// TwinCAT 3 PLC project Main
// ProgramVersion: 3.1.4023.0
// libraries:
//   Tc2_MC2, * (Beckhoff Automation GmbH)
//   Tc2_Standard, * (Beckhoff Automation GmbH)
//   Tc2_System, * (Beckhoff Automation GmbH)
//   Tc3_Module, * (Beckhoff Automation GmbH)
// project tree:
//   DUTs/Control/ ForceControlParam.TcDUT (not stored), JogParam.TcDUT (not stored)
//   DUTs/ MotorParam.TcDUT, MotorState.TcDUT (not stored), SystemControlMode.TcDUT (not stored), SystemControlParam.TcDUT
//   GVLs/ GVL.TcGVL (not stored)
//   / PlcTask.TcTTO
//   POUs/ MAIN.TcPOU, SystemControl.TcPOU
//   POUs/Safety/ VelocitySaturation.TcPOU
//   POUs/Converter/ CableVelocityToMotorAngularVelocity.TcPOU, MotorAngularVelocityToCableVelocity.TcPOU, MotorDegreeToCablePosition.TcPOU (not stored)
// real-time tasks:
//   TASK PlcTask: cycle T#10ms, priority 20, ADS port 350
// motion (NC):
//   TASK NC-Task 1 SAF: cycle T#2ms, priority 4, ADS port 501
//   TASK NC-Task 1 SVB: cycle T#10ms, priority 8, ADS port 511
//   AXIS Axis 1 (id 1)
//     General: UnitName=Degree
//     Dynamic: Acceleration=1080, Deceleration=1080, Jerk=3240
//     Velo: RefSearch=180, RefSync=180, SlowManual=180, FastManual=360, Fast=18075.9448242188, Maximum=720
//     PositionAreaControl: Enable=false
//     TargetPosControl: Enable=false
//     OtherSettings: AllowMotionCmdToSlave=true
//     encoder EncType=8
//       EncPara: ScaleFactorNumerator=360, ScaleFactorDenominator=1048576, MaxCount=#xffffffff
//     drive DrvType=9
//       DrvPara: MaxCount=#xffffffff, DriveControlDWord=#x00000100
//         Analog: VeloReferenz=360, VeloScale=1.02400649589962, TorqueSetpointScale=10, ScaleFactorActTorque=0.1
//         TimeComp: TaskDelayCycles=1
//     controller CtrType=1
//       CtrPara: PriorControlFactor=1
//         PosDiffControl: Enable=false
//         Observer: BandWidth=20
// I/O:
//   DEVICE Device 3 (EtherCAT), AmsNetId 192.168.137.1.4.1
//     Term 1 (EK1100) [EK1100 EtherCAT Coupler (2A E-Bus)]
//       Term 2 (EL9505) [EL9505 Power supply terminal 5V]
//       Term 3 (EL3356) [EL3356 1Ch. Ana. Input Resistor Bridge Terminal, 16bit, High Precision]
//       Term 5 (EL9011) [EL9011 End Terminal]
//     Drive 4 (AX5106-0000-0203) [AX5106-0000-0203 EtherCAT Drive (SoE, 1 Ch.)]
// variable links:
//   NC-Task 1 SAF/Axes/Axis 1 <-> Device 3 (EtherCAT)/Drive 4 (AX5106-0000-0203)
//     Drive/Inputs/In/nDcOutputTime <-> InfoData/DcOutputShift
//     Drive/Inputs/In/nState1 <-> AT/Drive status word @bit 8
//     Drive/Inputs/In/nState2 <-> AT/Drive status word
//     Drive/Inputs/In/nState4 @bit 1 <-> WcState/InputToggle
//     Drive/Inputs/In/nState4 <-> WcState/WcState
//     Drive/Outputs/Out/nCtrl1 <-> MDT/Master control word @bit 8
//     Enc/Inputs/In/nDcInputTime <-> InfoData/DcInputShift
//     Enc/Inputs/In/nState4 @bit 1 <-> WcState/InputToggle
//     Enc/Inputs/In/nState4 <-> WcState/WcState

CONFIGURATION Main
    RESOURCE PLC ON TwinCAT3
        TASK PlcTask(INTERVAL := T#10ms, PRIORITY := 20);
        PROGRAM MAIN WITH PlcTask : MAIN;
    END_RESOURCE
END_CONFIGURATION

// ---- DUTs/MotorParam.TcDUT
TYPE MotorParam :
STRUCT
	// 发送给电机的速度
	target_axis_velocity_raw : LREAL;
	
	// 期望的放绳速度
	target_cable_velocity : LREAL;
	
	// 最大最小速度(mm/s)
	max_cable_velocity : LREAL := 1000;
	min_cable_velocity : LREAL := -1000;
END_STRUCT
END_TYPE

// ---- DUTs/SystemControlParam.TcDUT
TYPE SystemControlParam :
STRUCT
	is_motor_poweron : BOOL;
	is_system_exit : BOOL;
	is_system_control : BOOL;
	system_control_mode : SystemControlMode;
	
	// Debug
	is_motor_jog : BOOL;
	jog_param : JogParam;
	// ConstForce
	is_force_control : BOOL;
	force_control_param : ForceControlParam;
END_STRUCT
END_TYPE

// ---- POUs/MAIN.TcPOU
PROGRAM MAIN
VAR
	SystemControl : SystemControl;
	
	system_control_param : SystemControlParam;
	motor_state : MotorState;
	motor_param : MotorParam;
END_VAR

// 系统状态读取
GVL.axis1.ReadStatus();
motor_state.is_motor_closedloop := GVL.axis1.Status.ControlLoopClosed;
motor_state.axis_position_raw := GVL.axis1.NcToPlc.ActPos;
motor_state.axis_velocity_raw := GVL.axis1.NcToPlc.ActVelo;

// 电机参数转换
MotorDegreeToCablePosition(motor_position:= motor_state.axis_position_raw, cable_position=> motor_state.cable_position);
MotorAngularVelocityToCableVelocity(motor_velocity:= motor_state.axis_velocity_raw, cable_velocity=> motor_state.cable_velocity);

// 控制状态机
SystemControl(
	motor_axis:= GVL.axis1, 
	system_control_param:= system_control_param, 
	motor_state:= motor_state, 
	target_velocity=> motor_param.target_cable_velocity);

// 安全限制 
VelocitySaturation(
	velocity:= motor_param.target_cable_velocity, 
	max_velocity:= motor_param.max_cable_velocity, 
	min_velocity:= motor_param.min_cable_velocity);

// 电机参数转换
CableVelocityToMotorAngularVelocity(cable_velocity:= motor_param.target_cable_velocity, motor_velocity=> motor_param.target_axis_velocity_raw);

END_PROGRAM

// ---- POUs/SystemControl.TcPOU
FUNCTION_BLOCK SystemControl
VAR_IN_OUT
	motor_axis : Tc2_MC2.AXIS_REF;
	system_control_param : SystemControlParam;
	motor_state : MotorState;
END_VAR
VAR_OUTPUT
	target_velocity : LREAL;
END_VAR
VAR
	motorPower : Tc2_MC2.MC_Power;
END_VAR

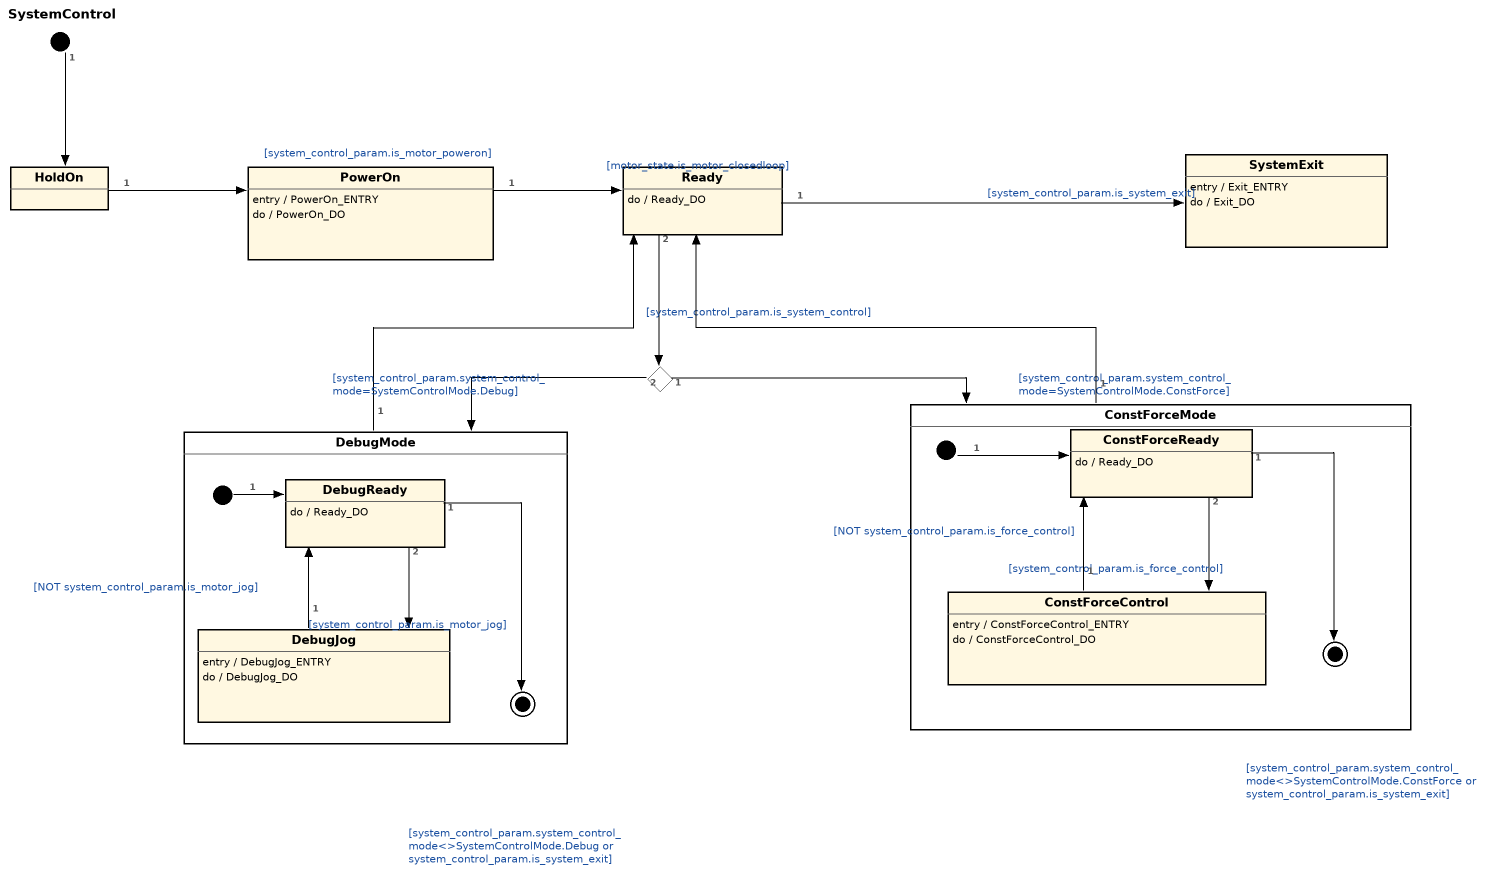
STATECHART SystemControl  // abortable
    START StartState1
    STATE HoldOn
    STATE PowerOn
        entry / PowerOn_ENTRY
        do / PowerOn_DO
    STATE Ready
        do / Ready_DO
    STATE SystemExit
        entry / Exit_ENTRY
        do / Exit_DO
    CHOICE ChoiceElement1
    COMPOSITE STATE ConstForceMode
        START StartState3
        STATE ConstForceReady
            do / Ready_DO
        STATE ConstForceControl
            entry / ConstForceControl_ENTRY
            do / ConstForceControl_DO
        END EndState2
        StartState3 -> ConstForceReady  // priority 1, on completion
        ConstForceReady -> EndState2 [system_control_param.system_control_mode<>SystemControlMode.ConstForce or system_control_param.is_system_exit] // priority 1
        ConstForceReady -> ConstForceControl [system_control_param.is_force_control] // priority 2
        ConstForceControl -> ConstForceReady [NOT system_control_param.is_force_control] // priority 1
    END_STATE
    COMPOSITE STATE DebugMode
        START StartState2
        STATE DebugReady
            do / Ready_DO
        STATE DebugJog
            entry / DebugJog_ENTRY
            do / DebugJog_DO
        END EndState1
        StartState2 -> DebugReady  // priority 1, on completion
        DebugReady -> EndState1 [system_control_param.system_control_mode<>SystemControlMode.Debug or system_control_param.is_system_exit] // priority 1
        DebugReady -> DebugJog [system_control_param.is_motor_jog] // priority 2
        DebugJog -> DebugReady [NOT system_control_param.is_motor_jog] // priority 1
    END_STATE
    StartState1 -> HoldOn  // priority 1, on completion
    HoldOn -> PowerOn [system_control_param.is_motor_poweron] // priority 1
    PowerOn -> Ready [motor_state.is_motor_closedloop] // priority 1
    Ready -> SystemExit [system_control_param.is_system_exit] // priority 1
    Ready -> ChoiceElement1 [system_control_param.is_system_control] // priority 2
    ChoiceElement1 -> ConstForceMode [system_control_param.system_control_mode=SystemControlMode.ConstForce] // priority 1
    ChoiceElement1 -> DebugMode [system_control_param.system_control_mode=SystemControlMode.Debug] // priority 2
    ConstForceMode -> Ready  // priority 1, on completion
    DebugMode -> Ready  // priority 1, on completion
END_STATECHART

ACTION ConstForceControl_DO:

END_ACTION

ACTION ConstForceControl_ENTRY:

END_ACTION

ACTION DebugJog_DO:
target_velocity := system_control_param.jog_param.jog_velocity;
END_ACTION

ACTION DebugJog_ENTRY:

END_ACTION

ACTION Exit_DO:
motorPower(
	Axis:= motor_axis, 
	Enable:= FALSE, 
	Enable_Positive:= TRUE, 
	Enable_Negative:= TRUE, 
	Override:= , 
	BufferMode:= , 
	Options:= , 
	Status=> , 
	Busy=> , 
	Active=> , 
	Error=> , 
	ErrorID=> );
END_ACTION

ACTION Exit_ENTRY:
target_velocity := 0;
END_ACTION

ACTION PowerOn_DO:
motorPower(
	Axis:= motor_axis, 
	Enable:= TRUE, 
	Enable_Positive:= TRUE, 
	Enable_Negative:= TRUE, 
	Override:= , 
	BufferMode:= , 
	Options:= , 
	Status=> , 
	Busy=> , 
	Active=> , 
	Error=> , 
	ErrorID=> );
END_ACTION

ACTION PowerOn_ENTRY:

END_ACTION

ACTION Ready_DO:
target_velocity := 0;
END_ACTION

END_FUNCTION_BLOCK

// ---- POUs/Converter/MotorAngularVelocityToCableVelocity.TcPOU
FUNCTION MotorAngularVelocityToCableVelocity : LREAL
VAR_INPUT
	motor_velocity : LREAL;
END_VAR
VAR_OUTPUT
	cable_velocity : LREAL;
END_VAR
VAR
END_VAR

cable_velocity := motor_velocity;

END_FUNCTION

// ---- POUs/Safety/VelocitySaturation.TcPOU
FUNCTION VelocitySaturation : LREAL
VAR_IN_OUT
	velocity : LREAL;
	max_velocity : LREAL;
	min_velocity : LREAL;
END_VAR
VAR
	velocity_sign : LREAL;
END_VAR

IF velocity >= 0 THEN
	velocity_sign := 1;
ELSE
	velocity_sign := -1;
END_IF

IF ABS(velocity) > max_velocity THEN
	velocity := max_velocity * velocity_sign;
END_IF
IF ABS(velocity) < min_velocity THEN
	velocity := min_velocity * velocity_sign;
END_IF

END_FUNCTION

// ---- POUs/Converter/CableVelocityToMotorAngularVelocity.TcPOU
FUNCTION CableVelocityToMotorAngularVelocity : LREAL
VAR_INPUT
	cable_velocity : LREAL;
END_VAR
VAR_OUTPUT
	motor_velocity : LREAL;
END_VAR
VAR
END_VAR

motor_velocity := cable_velocity;

END_FUNCTION
